(* IEC 61131-3 sources: go-st/tests, 9 files *)

(* ---- 001_simpliest.st ---- *)
PROGRAM simpliest
  VAR
    /*
        просто объявление переменных, без каких либо вычислений
        + многострочный комментарий
    */
    i : INT := 5;
    j : INT; // проверка, что значения по умолчанию может не быть + комментарий
    (*
        проверка, что поддерживаются значения со знаком
        + многострочный комментарий
    *)
    k : INT := -42;
  END_VAR

  i := 15;
  // k := uv; // раскомментировать для ошибки
END_PROGRAM

(* ---- 002_arithmetic.st ---- *)
PROGRAM arithmetic
  VAR
    i : INT;
    j : INT;
    k : INT := 42;
  END_VAR

  i := 15+j;
  j := 5 + 2*i*(30-i)/5; // проверка приоритета арифмитических операций
  k := k + -2;           // проверка, что унарный минус отработает
END_PROGRAM

(* ---- 003_iftest.st ---- *)
PROGRAM iftest
  VAR
    i       : INT;
    divisor : INT;
    mult    : INT;
    test    : INT;
  END_VAR

  i := i+1;
  IF i MOD 5 = 0 THEN
    divisor := 5;
    IF i/5 = 1 THEN    // тест условия внутри условия
      mult := 1;
    ELSIF i/5 = 2 THEN // тест блока ELSIF
      mult := 2;
    ELSE               // тест блока ELSE
      mult := 3;
    END_IF
  ELSIF i MOD 4 = 0 THEN
    divisor := 4;
    mult := i/4;
  ELSIF i MOD 3 = 0 THEN
    divisor := 3;
    mult := i/3;
  ELSIF i MOD 2 = 0 THEN
    divisor := 2;
    mult := i/2;
  ELSIF i MOD 1 = 0 THEN
    divisor := 1;
    mult := i;
  // тест условия c ELSIF без ELSE
  END_IF

  // тест простого условия без ELSE
  IF mult <> 1 THEN
    test := mult*divisor;
  END_IF
END_PROGRAM

(* ---- 004_parse_err.st ---- *)
PROGRAM simpliest
  VAR
    i : INT := 5;
  END_VAR
  i := 1x5;
END_PROGRAM

(* ---- 005_cast.st ---- *)
PROGRAM cast
  VAR
    i8   : SINT;
    i16  : INT;
    i32  : DINT;
    i64  : LINT;
    ui8  : USINT;
    ui16 : UINT;
    ui32 : UDINT;
    ui64 : ULINT;
    test : INT;
  END_VAR

  test := test + 1;
  IF test = 1 THEN
    // max unsigned
    i8 := i8-1;
    i16 := i16-1;
    i32 := i32-1;
    i64 := i64-1;
    ui8 := ui8-1;
    // ui8 := ui16-1; // если раскомментировать, можно увидеть ошибку
    ui16 := ui16-1;
    ui32 := ui32-1;
    ui64 := ui64-1;
    // i8 := i8 + ui64; // если раскомментировать, можно увидеть ошибку
  ELSIF test = 2 THEN
    // max signed
    i8 := 16#7F;
    i16 := 16#7FFF;
    i32 := 16#7FFF_FFFF;
    i64 := 16#7FFF_FFFF_FFFF_FFFF;
  ELSIF test = 3 THEN
    // max signed
    i8 := i8 + 1;
    i16 := i16 + 1;
    i32 := i32 + 1;
    i64 := i64 + 1;
    ui16 := INT_TO_UINT(i16);
    // ui16 := DINT_TO_UINT(i16); // если раскомментировать, можно увидеть ошибку
  END_IF
END_PROGRAM

(* ---- 006_floats.st ---- *)
PROGRAM cast
  VAR
    f1 : REAL := 1;
    f2 : LREAL := -0.5;
    f3 : REAL := 5.E1;
    test: INT;
  END_VAR
  test := test + 1;
  IF test = 1 THEN
    // f1 := f2; // ошибка каста
    f1 := LREAL_TO_REAL(f2);
    f2 := f3; // скрытый каст
  ELSIF test = 2 THEN
    f3 := f1 * 2; // -0,5*2=-1
    f2 := f1 + f3;  // -0,5+-1 = -1,5
  ELSIF test = 3 THEN
    f2 := f3/f1-f2; // -1/-0,5 - -1,5 = 3,5
  END_IF
END_PROGRAM

(* ---- 007_while.st ---- *)
PROGRAM while_test
  VAR
    i : INT;
    counter : INT;
    r : INT;
    r2 : INT;
  END_VAR
  WHILE i<5 DO
    r := r+i;
    i := i+1;
  END_WHILE
  i := i-3;

  // ===== ТЕСТ: WHILE с CONTINUE (пропуск итерации) =====
  counter := 0;
  r2 := 0;
  WHILE counter < 5 DO
      counter := counter + 1;
      IF counter MOD 2 = 0 THEN
          CONTINUE; // Пропускаем четные числа
      END_IF;
      r2 := r2 + counter; // Суммируем только нечетные
  END_WHILE;

  // ===== ТЕСТ: WHILE с EXIT =====
  counter := 0;
  WHILE counter < 10 DO
      counter := counter + 1;
      IF counter >= 7 THEN
          EXIT; // Выходим после 7 итераций
      END_IF;
  END_WHILE;
END_PROGRAM

(* ---- 008_func.st ---- *)
PROGRAM FunctionTest
  VAR
    in         : INT;
    square     : INT;
    factorial  : INT;
    factorial6 : INT;
  END_VAR

  in := 5;
  square := Square(in);
  factorial := Factorial(in);
  factorial6 := Factorial(6);
END_PROGRAM

// Функция вычисления квадрата числа
FUNCTION Square : INT
  VAR_INPUT
    num : INT;
  END_VAR
    Square := num * num;
END_FUNCTION

// // Функция вычисления факториала (рекурсивная)
// FUNCTION FactorialRecurce : INT
//   VAR_INPUT
//     n : INT;
//   END_VAR
//   VAR
//     temp : INT;
//   END_VAR
//     IF n <= 1 THEN
//         Factorial := 1;
//     ELSE
//         Factorial := n * FactorialRecurce(n - 1);
//     END_IF
// END_FUNCTION

FUNCTION Factorial : INT
VAR_INPUT
    n : INT;
END_VAR
VAR
    result : INT := 1;
    i : INT;
END_VAR
    FOR i := 1 TO n BY 1 DO
        result := result * i;
    END_FOR
    Factorial := result;
END_FUNCTION

(* ---- 009_for.st ---- *)
PROGRAM ForTest
  VAR
    v : REAL;
    i : REAL;
  END_VAR

  FOR i := 10 TO 8 BY -0.5 DO
    v := v + i; // 10+9.5+9+8.5+8=45
  END_FOR
END_PROGRAM
